FUNCTION_BLOCK LRAnalog (* Composite FB wrapping other FBs *)
  (* Standard: 61499-2 *)
  (* Version 1.0, 2021-03-18, AK120569 *)
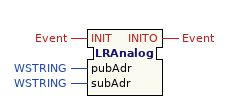
  EVENT_INPUT
    INIT; (* Initialization Request *)
  END_EVENT
  EVENT_OUTPUT
    INITO; (* Initialization Confirm *)
  END_EVENT
  VAR_INPUT
    pubAdr : WSTRING;
    subAdr : WSTRING;
  END_VAR
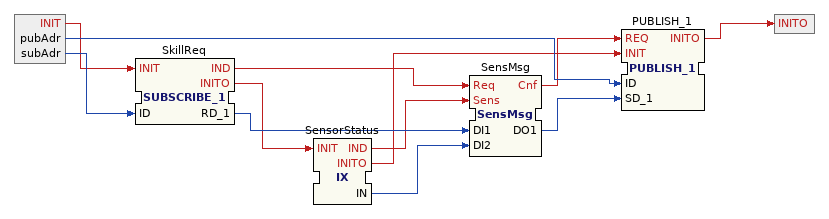
  FBS
    SkillReq : SUBSCRIBE_1;
    SensorStatus : IX;
    PUBLISH_1 : PUBLISH_1;
    SensMsg : SensMsg;
  END_FBS
  EVENT_CONNECTIONS
    INIT TO SkillReq.INIT;
    SkillReq.IND TO SensMsg.Req;
    SensorStatus.IND TO SensMsg.Sens;
    SensMsg.Cnf TO PUBLISH_1.REQ;
    SkillReq.INITO TO SensorStatus.INIT;
    SensorStatus.INITO TO PUBLISH_1.INIT;
    PUBLISH_1.INITO TO INITO;
  END_CONNECTIONS
  DATA_CONNECTIONS
    pubAdr TO PUBLISH_1.ID;
    subAdr TO SkillReq.ID;
    SkillReq.RD_1 TO SensMsg.DI1;
    SensMsg.DO1 TO PUBLISH_1.SD_1;
    SensorStatus.IN TO SensMsg.DI2;
  END_CONNECTIONS
END_FUNCTION_BLOCK
